PROGRAM MAIN
VAR
END_VAR

POU();

END_PROGRAM

(* stored: Version 1.1.0.1, ProductVersion 3.1.4024.3
   POU MAIN: Id {363fe7e3-f3b9-4a70-a512-6dd415481581}, SpecialFunc None *)
